// TIA Portal V21 export
FUNCTION_BLOCK "VesselLamp"   // FB7, LAD
{ S7_Optimized_Access := 'FALSE' }
// stored: AutoNumber false, SetENOAutomatically false
   VAR_INPUT
      Secs : Bool;
      AlwaysTrue : Bool;
      AlwaysFalse : Bool;
   END_VAR
   VAR_OUTPUT
      DONE_BIT : Bool;
      ES_MINIT : DInt;
      ES_SEC : DInt;
   END_VAR
   VAR
      LF01 { S7_SetPoint := 'True'} : "TIMER";   // LF01
   END_VAR
BEGIN

REGION Network 1: #VslLamp01
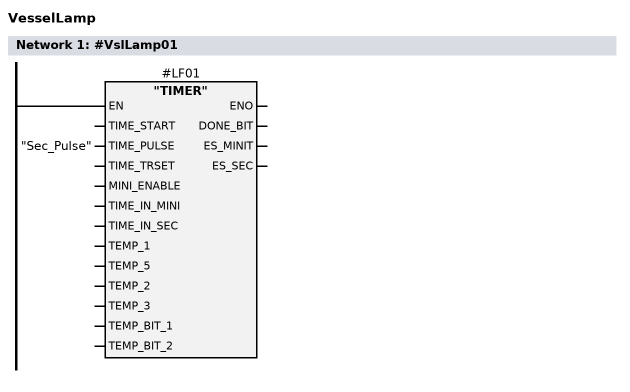
   RUNG wire#powerrail
      #LF01(TIME_START :=, TIME_PULSE := "Sec_Pulse", TIME_TRSET :=, MINI_ENABLE :=, TIME_IN_MINI :=, TIME_IN_SEC :=, TEMP_1 :=, TEMP_5 :=, TEMP_2 :=, TEMP_3 :=, TEMP_BIT_1 :=, TEMP_BIT_2 :=, DONE_BIT =>, ES_MINIT =>, ES_SEC =>)
   END_RUNG
   // the same network as SCL:
   #LF01(TIME_PULSE := "Sec_Pulse");   // "TIMER"
END_REGION
END_FUNCTION_BLOCK
